// TIA Portal V20 export
// export: Created 2025-12-01T14:57:06.202476Z, ExportSetting None, DisplayName Totally Integrated Automation Portal, DisplayVersion V20 Update 3, DisplayName TIA Portal Openness, DisplayVersion V20 Update 3, DisplayName TIA Portal Version Control Interface, DisplayVersion V20 Update 3, DisplayName STEP 7 Professional, DisplayVersion V20 Update 3, DisplayName STEP 7 Safety, DisplayVersion V20 Update 2, DisplayName WinCC Basic/Comfort/Advanced, DisplayVersion V20 Update 3, DisplayName WinCC Professional, DisplayVersion V20 Update 3, DisplayName WinCC Unified, DisplayVersion V20 Update 3
FUNCTION "FC910_CNT_pulsos_UHS" : Void   // FC910, LAD
{ S7_Optimized_Access := 'FALSE' }
AUTHOR : GENERAL
NAME : 20130301
VERSION : 3.0
// stored: AutoNumber false, SetENOAutomatically false
   VAR_INPUT
      CUENTA_UP : Bool;
      RESET : Bool;
      Valor_Cuenta : UDInt;
   END_VAR
   VAR_OUTPUT
      Cuenta_OK : Bool;
   END_VAR
   VAR_IN_OUT
      Valor_Actual : UDInt;
   END_VAR
   VAR_TEMP
      TEMP_Cuenta_OK : Bool;
   END_VAR
BEGIN

REGION Network 1
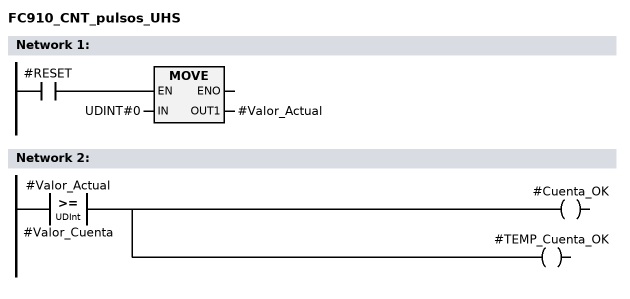
   RUNG wire#powerrail
      Contact( #RESET )
      { S7_GenerateENO := "TRUE" } Move(in := UDINT#0, out1 => #Valor_Actual)
   END_RUNG
   // the same network as SCL:
   IF #RESET THEN #Valor_Actual := UDINT#0; END_IF;
END_REGION

REGION Network 2
   RUNG wire#powerrail
      { S7_Templates := "SrcType := UDInt" } GE_Contact(in1 := #Valor_Actual, in2 := #Valor_Cuenta)
      wire#w1
      Coil( #Cuenta_OK )
   END_RUNG
   RUNG wire#w1
      Coil( #TEMP_Cuenta_OK )
   END_RUNG
   // the same network as SCL:
   #Cuenta_OK := #Valor_Actual >= #Valor_Cuenta;
   #TEMP_Cuenta_OK := #Cuenta_OK;
END_REGION

NETWORK
TITLE = 
      A     #CUENTA_UP;
      AN    #TEMP_Cuenta_OK;
      JNB   _002;
      L     #Valor_Actual;
      L     1;
      +D;
      T     #Valor_Actual;
_002: NOP   0;
END_FUNCTION
